{attribute addProperty BoxType "EP7041-0002-0016"}
{attribute addProperty Id "StatusAT %I*Status_1C57BC2B516.375"}
{attribute addProperty CRC "1113461332"}
{attribute addProperty SizeInBites "51"}
{attribute addProperty SizeInBytes "6.375"}
TYPE STM_Status_425E1254 :
STRUCT
	{attribute addProperty Name "Status"}
	Status AT %I* : Status_1C57BC2B;
END_STRUCT
END_TYPE

(* stored: Version 1.2.0.0, ProductVersion 3.1.4024.9
   DUT STM_Status_425E1254: Id {36610edc-7ae1-4725-ab93-b08b3a0a7dc7} *)
